(*

## Short summary
This interface provides assert statements for 32 bit ``TIME``  

.. <legal notes>

legal notes
=================
| SPDX-FileCopyrightText: © 2022 ekvip automation GmbH <info@ekvip.de>
| SPDX-License-Identifier: Apache-2.0
| For details check: Apache-2.0_

.. _Apache-2.0: https://www.apache.org/licenses/LICENSE-2.0

.. </legal notes>



*)

INTERFACE I32BitTimeAssertions EXTENDS __SYSTEM.IQueryInterface

(*

## Short summary
This assertion method checks whether time has elapsed since the timestamp time

.. <legal notes>

legal notes
=================
| SPDX-FileCopyrightText: © 2022 ekvip automation GmbH <info@ekvip.de>
| SPDX-License-Identifier: Apache-2.0
| For details check: Apache-2.0_

.. _Apache-2.0: https://www.apache.org/licenses/LICENSE-2.0

.. </legal notes>



*)

METHOD timeHasExpired
VAR_INPUT
	(* start time you get it with ``TIME()`` *)
	timestamp		:TIME;
	(* timeout like ``t#300ms`` *)
	expiringTime	:TIME;
	(* message if the assertion is false *)
	message			:AssertMessage;
END_VAR
END_METHOD

(*

## Short summary
This assertion method checks that the time since the timestamp time has not yet elapsed

.. <legal notes>

legal notes
=================
| SPDX-FileCopyrightText: © 2022 ekvip automation GmbH <info@ekvip.de>
| SPDX-License-Identifier: Apache-2.0
| For details check: Apache-2.0_

.. _Apache-2.0: https://www.apache.org/licenses/LICENSE-2.0

.. </legal notes>



*)

METHOD timeHasNotExpired
VAR_INPUT
	(* start time you get it with ``TIME()`` *)
	timestamp		:TIME;
	(* timeout like ``t#300ms`` *)
	expiringTime	:TIME;
	(* message if the assertion is false *)
	message			:AssertMessage;
END_VAR
END_METHOD

(*

## Short summary
This assertion method checks if the current value is equal to the expected value

.. <legal notes>

legal notes
=================
| SPDX-FileCopyrightText: © 2022 ekvip automation GmbH <info@ekvip.de>
| SPDX-License-Identifier: Apache-2.0
| For details check: Apache-2.0_

.. _Apache-2.0: https://www.apache.org/licenses/LICENSE-2.0

.. </legal notes>



*)

METHOD valueIsEqualTo
VAR_INPUT
	(* current value to check *)
	currentValue	:TIME;
	(* expected value to compare *)
	expectedValue	:TIME;
	(* message if the assertion is false *)
	message			:AssertMessage;
END_VAR
END_METHOD

(*

## Short summary
This assertion method checks if the current value is greater than the less value

.. <legal notes>

legal notes
=================
| SPDX-FileCopyrightText: © 2022 ekvip automation GmbH <info@ekvip.de>
| SPDX-License-Identifier: Apache-2.0
| For details check: Apache-2.0_

.. _Apache-2.0: https://www.apache.org/licenses/LICENSE-2.0

.. </legal notes>



*)

METHOD valueIsGreaterThan
VAR_INPUT
	(* current value to check *)
	currentValue	:TIME;
	(* less than lower limit *)
	lessValue		:TIME;
	(* message if the assertion is false *)
	message			:AssertMessage;
END_VAR
END_METHOD

(*

## Short summary
This assertion method checks if the current value is inside a limit

**Attention:** 
	limits are included: ``valueIsInRangeOf(t#3ms,t#3ms ,t#3ms)`` is a true assertion

.. <legal notes>

legal notes
=================
| SPDX-FileCopyrightText: © 2022 ekvip automation GmbH <info@ekvip.de>
| SPDX-License-Identifier: Apache-2.0
| For details check: Apache-2.0_

.. _Apache-2.0: https://www.apache.org/licenses/LICENSE-2.0

.. </legal notes>



*)

METHOD valueIsInRangeOf
VAR_INPUT
	(* lower limit for the current value *)
	lowerLimit		:TIME;
	(* current value to check *)
	currentValue	:TIME;
	(* upper limit for the current value *)
	upperLimit		:TIME;
	(* message if the assertion is false *)
	message			:AssertMessage;
END_VAR
END_METHOD

(*

## Short summary
This assertion method checks if the current value is less than the greater value

.. <legal notes>

legal notes
=================
| SPDX-FileCopyrightText: © 2022 ekvip automation GmbH <info@ekvip.de>
| SPDX-License-Identifier: Apache-2.0
| For details check: Apache-2.0_

.. _Apache-2.0: https://www.apache.org/licenses/LICENSE-2.0

.. </legal notes>



*)

METHOD valueIsLessThan
VAR_INPUT
	(* current value to check *)
	currentValue	:TIME;
	(* greater than upper limit *)
	greaterValue	:TIME;
	(* message if the assertion is false *)
	message			:AssertMessage;
END_VAR
END_METHOD

(*

## Short summary
This assertion method checks if the current value is less than or equal to the maximum value

.. <legal notes>

legal notes
=================
| SPDX-FileCopyrightText: © 2022 ekvip automation GmbH <info@ekvip.de>
| SPDX-License-Identifier: Apache-2.0
| For details check: Apache-2.0_

.. _Apache-2.0: https://www.apache.org/licenses/LICENSE-2.0

.. </legal notes>



*)

METHOD valueIsMax
VAR_INPUT
	(* current value to check *)
	currentValue	:TIME;
	(* upper limit for the current value *)
	maximumValue	:TIME;
	(* message if the assertion is false *)
	message			:AssertMessage;
END_VAR
END_METHOD

(*

## Short summary
This assertion method checks if the current value is greater than or equal to the minimum value

.. <legal notes>

legal notes
=================
| SPDX-FileCopyrightText: © 2022 ekvip automation GmbH <info@ekvip.de>
| SPDX-License-Identifier: Apache-2.0
| For details check: Apache-2.0_

.. _Apache-2.0: https://www.apache.org/licenses/LICENSE-2.0

.. </legal notes>



*)

METHOD valueIsMin
VAR_INPUT
	(* current value to check *)
	currentValue	:TIME;
	(* lower limit for the current value *)
	minimumValue	:TIME;
	(* message if the assertion is false *)
	message			:AssertMessage;
END_VAR
END_METHOD

(*

## Short summary
This assertion method checks if the current value is not equal to the unexpected value

.. <legal notes>

legal notes
=================
| SPDX-FileCopyrightText: © 2022 ekvip automation GmbH <info@ekvip.de>
| SPDX-License-Identifier: Apache-2.0
| For details check: Apache-2.0_

.. _Apache-2.0: https://www.apache.org/licenses/LICENSE-2.0

.. </legal notes>



*)

METHOD valueIsNotEqualTo
VAR_INPUT
	(* current value to check *)
	currentValue	:TIME;
	(* unexpected value to compare *)
	unexpectedValue	:TIME;
	(* message if the assertion is false *)
	message			:AssertMessage;
END_VAR
END_METHOD

END_INTERFACE

(* stored: Version 1.1.0.1, ProductVersion 3.1.4024.11
   Itf I32BitTimeAssertions: Id {60a6b4d0-df96-4aeb-8481-d17b2fcabbc6}
   Method timeHasExpired: Id {12c8930a-0817-4ba5-94c9-02085621151d}
   Method timeHasNotExpired: Id {bbc0d366-91eb-492d-a0ac-86add5f20281}
   Method valueIsEqualTo: Id {4ca608a3-02a1-4ff6-8dea-1d8702a682b2}
   Method valueIsGreaterThan: Id {da23d5c2-8c3b-41c2-a2f4-ddddb4882514}
   Method valueIsInRangeOf: Id {639c1b45-ac85-4489-8c40-7131638a0109}
   Method valueIsLessThan: Id {aa83ad34-4d02-4acb-b55d-8ca7a5f0d96d}
   Method valueIsMax: Id {a2709032-f6be-4ad1-9c85-51ea5ba49468}
   Method valueIsMin: Id {05be0ec3-33be-4e62-8fd0-740b873a69ed}
   Method valueIsNotEqualTo: Id {6e11fb94-b2d8-4ccd-9d10-b3165c83bb90} *)
